Staubli VAL3: insertItem.pgx

public program insertItem(InstrItem& x_sItem[] (dimensions=1), num x_nIndex (dimensions=1))
  local num l_sItem
begin
  if x_nIndex<=0
    x_nIndex=0
  else
    insert(pEdit.iEvent[x_nIndex])
  endIf
  call setItem(x_sItem,x_nIndex)
end
